// TIA Portal V20 export
DATA_BLOCK "Config"   // DB48
// stored: Access Published, MemoryReserve 100, Namespace Unit1.Em5
   VAR
      em : "LAF_typeEmConfiguration";
      axis : Array[0.._.U1EM5_NO_OF_AXES] of DB_ANY;
      cmTransferPnPLeftSafetyPin : "LBC_typeDigitalSignalConfiguration";
      cmTransferPnPLeftJRDetect : "LBC_typeDigitalSignalConfiguration";
      cmTransferPnPRightSafetyPin : "LBC_typeDigitalSignalConfiguration";
      cmTransferPnPRightJRDetect : "LBC_typeDigitalSignalConfiguration";
   END_VAR
   VAR RETAIN
      cmTransferPnPLeftAxisX : "LBC_typeAxis64PosConfiguration";
      cmTransferPnPLeftAxisY : "LBC_typeAxis64PosConfiguration";
      cmTransferPnPLeftAxisZ : "LBC_typeAxis64PosConfiguration";
      cmTransferPnPRightAxisX : "LBC_typeAxis64PosConfiguration";
      cmTransferPnPRightAxisY : "LBC_typeAxis64PosConfiguration";
      cmTransferPnPRightAxisZ : "LBC_typeAxis64PosConfiguration";
   END_VAR
   VAR
      cmTransferPnPLeftClampOpenClose : "LBC_typeTwoWayActuatorConfiguration";
      cmTransferPnPRightClampOpenClose : "LBC_typeTwoWayActuatorConfiguration";
      softcam : Struct
         TransferPnPLeftAxisX : "LER_typeSoftCamInterface";
         TransferPnPLeftAxisY : "LER_typeSoftCamInterface";
         TransferPnPLeftAxisZ { S7_SetPoint := 'True'} : "LER_typeSoftCamInterface";
         TransferPnPRightAxisX { S7_SetPoint := 'True'} : "LER_typeSoftCamInterface";
         TransferPnPRightAxisY { S7_SetPoint := 'True'} : "LER_typeSoftCamInterface";
         TransferPnPRightAxisZ { S7_SetPoint := 'True'} : "LER_typeSoftCamInterface";
      END_STRUCT;
   END_VAR
BEGIN
   em.referenceDesignator.parent := WSTRING#'U1';
   em.referenceDesignator.relative := WSTRING#'EM0';
   cmTransferPnPLeftAxisX.referenceDesignator := WSTRING#'TRANSFER P&P LEFT X-Axis';
   cmTransferPnPLeftAxisY.referenceDesignator := WSTRING#'TRANSFER P&P LEFT Y-Axis';
   cmTransferPnPLeftAxisZ.referenceDesignator := WSTRING#'TRANSFER P&P LEFT Z-Axis';
   cmTransferPnPRightAxisX.referenceDesignator := WSTRING#'TRANSFER P&P RIGHT X-Axis';
   cmTransferPnPRightAxisY.referenceDesignator := WSTRING#'TRANSFER P&P RIGHT Y-Axis';
   cmTransferPnPRightAxisZ.referenceDesignator := WSTRING#'TRANSFER P&P RIGHT Z-Axis';
   cmTransferPnPLeftClampOpenClose.referenceDesignator := WSTRING#'P&P CLAMP LEFT';
   cmTransferPnPLeftClampOpenClose.monitoringDiscrepancy := T#5s;
   cmTransferPnPRightClampOpenClose.referenceDesignator := WSTRING#'P&P CLAMP RIGHT';
   cmTransferPnPRightClampOpenClose.monitoringDiscrepancy := T#5s;
END_DATA_BLOCK
